// LS Electric XG5000 project: 파이썬PLC485통신
// PLC LSPLC

PROGRAM NewProgram (task: 스캔 프로그램)

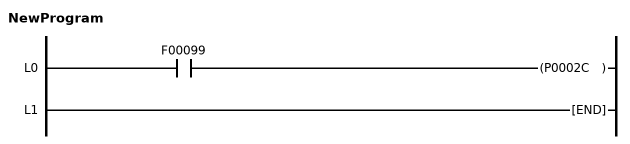
; L0
LOAD      F00099
OUT       P0002C
; L1
END